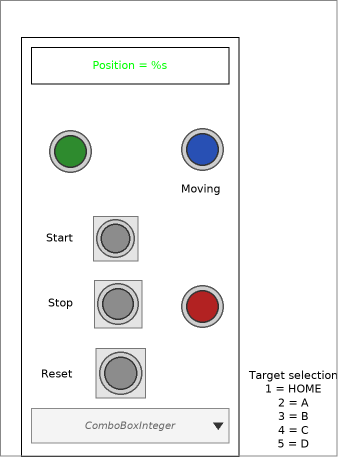
VISUALIZATION Visualization  // 338x457
    Rectangle (21,37 218x420)
    PushSwitch (93,280 50x48), variable: GVL_CTRL.xStopPB, behaviour: TAP, style: Switch-PushSwitch-Gray
    PushSwitch (93,348 55x50), variable: GVL_CTRL.xResetPB, behaviour: TAP, style: Switch-PushSwitch-Gray
    Label (31,359 52x30), "Reset"
    Label (38,288 45x30), "Stop"
    PushSwitch (93,214 45x49), variable: GVL_CTRL.xStartPB, behaviour: TAP, style: Switch-PushSwitch-Gray
    Label (31,223 57x30), "Start"
    Lamp1 (46,120 49x63), variable: GVL_CTRL.xReadyLamp, style: Lamp-Lamp1-Green
    Lamp1 (178,120 49x59), variable: GVL_CTRL.xMovingLamp, style: Lamp-Lamp1-Blue
    Label (126,174 150x30), "Moving"
    Lamp1 (178,280 49x53), variable: GVL_CTRL.xStopLamp, style: Lamp-Lamp1-Red
    Rectangle (31,47 198x37), "Position = %s", text variable: GVL.iiAtPos
    ComboBoxInteger (31,408 198x35), variable: GVL_CTRL.iTarget
    Label (249,362 89x95), "Target selection 1 = HOME 2 = A 3 = B 4 = C 5 = D"
END_VISUALIZATION

(* stored: Version 1.1.0.1
   Visu Visualization: Id {60ccff64-eff1-46b7-8302-bb69333e9ec5} *)
